% RSLogix 500 project inventoryManagement.RSS, saved by version 8.30.00.16 %
PROJECT "UNTITLED"    % processor: Bul.1763 MicroLogix 1100 Series B %

PROGRAM FILES
  LAD 2   24 rungs

DATA FILES
  O0 OUTPUT  4 elements
  I1 INPUT  6 elements
  S2 STATUS  66 elements
  B3 BINARY  1 elements
  T4 TIMER  1 elements
  C5 COUNTER  1 elements
  R6 CONTROL  1 elements
  N7 INTEGER  9 elements
  F8 FLOAT  1 elements
  ST9 BARCODE  10 elements

LADDER 2
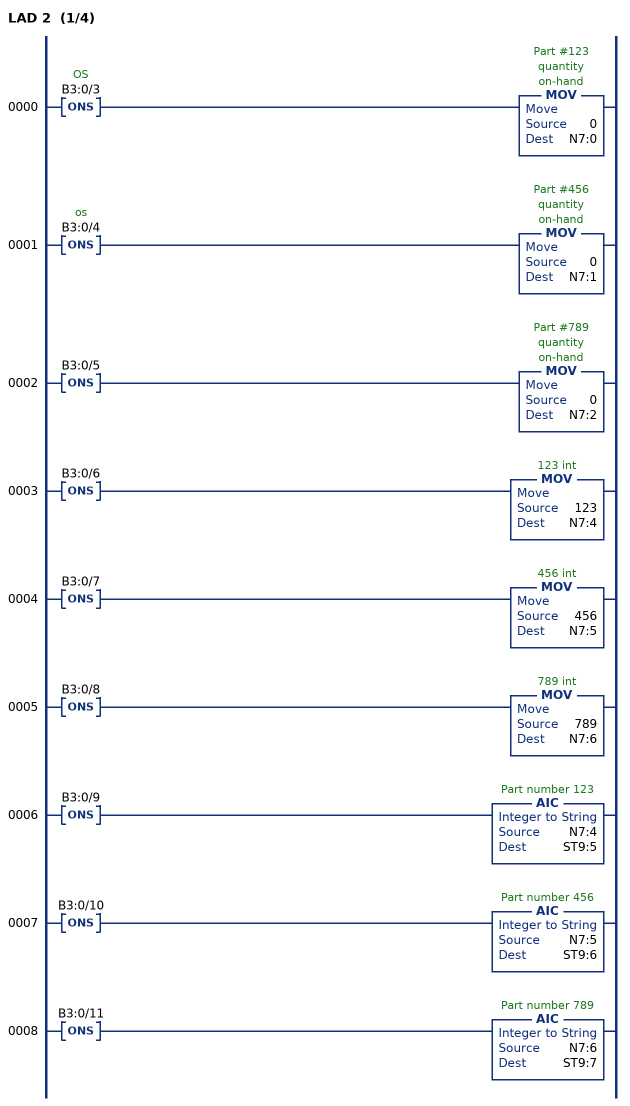
% Rung: 0 %
SOR ONS B3:0/3 MOV 0 N7:0 EOR
%   B3:0/3  "OS" %
%   N7:0  "Part #123 quantity on-hand" %
% Rung: 1 %
SOR ONS B3:0/4 MOV 0 N7:1 EOR
%   B3:0/4  "os" %
%   N7:1  "Part #456 quantity on-hand" %
% Rung: 2 %
SOR ONS B3:0/5 MOV 0 N7:2 EOR
%   N7:2  "Part #789 quantity on-hand" %
% Rung: 3 %
SOR ONS B3:0/6 MOV 123 N7:4 EOR
%   N7:4  "123 int" %
% Rung: 4 %
SOR ONS B3:0/7 MOV 456 N7:5 EOR
%   N7:5  "456 int" %
% Rung: 5 %
SOR ONS B3:0/8 MOV 789 N7:6 EOR
%   N7:6  "789 int" %
% Rung: 6 %
SOR ONS B3:0/9 AIC N7:4 ST9:5 EOR
%   N7:4  "123 int" %
%   ST9:5  "Part number 123" %
% Rung: 7 %
SOR ONS B3:0/10 AIC N7:5 ST9:6 EOR
%   N7:5  "456 int" %
%   ST9:6  "Part number 456" %
% Rung: 8 %
SOR ONS B3:0/11 AIC N7:6 ST9:7 EOR
%   N7:6  "789 int" %
%   ST9:7  "Part number 789" %

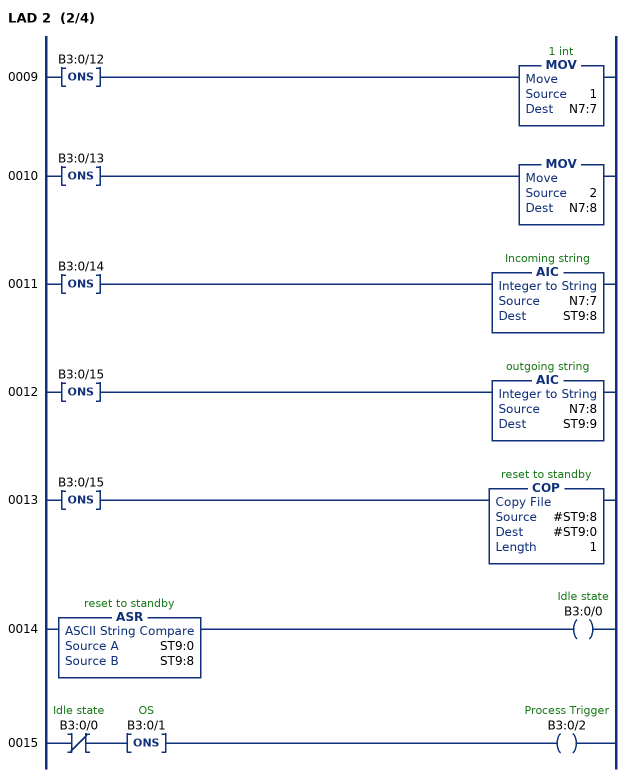
% Rung: 9 %
SOR ONS B3:0/12 MOV 1 N7:7 EOR
%   N7:7  "1 int" %
% Rung: 10 %
SOR ONS B3:0/13 MOV 2 N7:8 EOR
% Rung: 11 %
SOR ONS B3:0/14 AIC N7:7 ST9:8 EOR
%   N7:7  "1 int" %
%   ST9:8  "Incoming string" %
% Rung: 12 %
SOR ONS B3:0/15 AIC N7:8 ST9:9 EOR
%   ST9:9  "outgoing string" %
% Rung: 13 %
SOR ONS B3:0/15 COP #ST9:8 #ST9:0 1 EOR
%   ST9:8  "Incoming string" %
%   ST9:0  "reset to standby" %
% Rung: 14 %
SOR ASR ST9:0 ST9:8 OTE B3:0/0 EOR
%   ST9:0  "reset to standby" %
%   ST9:8  "Incoming string" %
%   B3:0/0  "Idle state" %
% Rung: 15 %
SOR XIO B3:0/0 ONS B3:0/1 OTE B3:0/2 EOR
%   B3:0/0  "Idle state" %
%   B3:0/1  "OS" %
%   B3:0/2  "Process Trigger" %

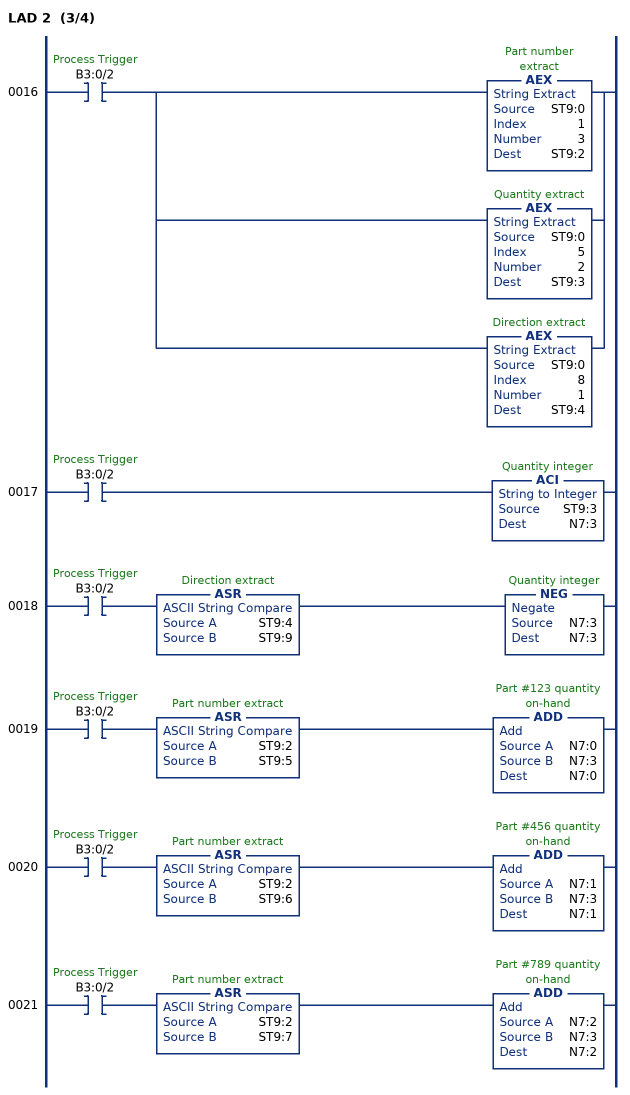
% Rung: 16 %
SOR XIC B3:0/2 BST AEX ST9:0 1 3 ST9:2 NXB BST AEX ST9:0 5 2 ST9:3 NXB AEX ST9:0 8 1 ST9:4 BND BND EOR
%   B3:0/2  "Process Trigger" %
%   ST9:0  "reset to standby" %
%   ST9:2  "Part number extract" %
%   ST9:3  "Quantity extract" %
%   ST9:4  "Direction extract" %
% Rung: 17 %
SOR XIC B3:0/2 ACI ST9:3 N7:3 EOR
%   B3:0/2  "Process Trigger" %
%   ST9:3  "Quantity extract" %
%   N7:3  "Quantity integer" %
% Rung: 18 %
SOR XIC B3:0/2 ASR ST9:4 ST9:9 NEG N7:3 N7:3 EOR
%   B3:0/2  "Process Trigger" %
%   ST9:4  "Direction extract" %
%   ST9:9  "outgoing string" %
%   N7:3  "Quantity integer" %
% Rung: 19 %
SOR XIC B3:0/2 ASR ST9:2 ST9:5 ADD N7:0 N7:3 N7:0 EOR
%   B3:0/2  "Process Trigger" %
%   ST9:2  "Part number extract" %
%   ST9:5  "Part number 123" %
%   N7:0  "Part #123 quantity on-hand" %
%   N7:3  "Quantity integer" %
% Rung: 20 %
SOR XIC B3:0/2 ASR ST9:2 ST9:6 ADD N7:1 N7:3 N7:1 EOR
%   B3:0/2  "Process Trigger" %
%   ST9:2  "Part number extract" %
%   ST9:6  "Part number 456" %
%   N7:1  "Part #456 quantity on-hand" %
%   N7:3  "Quantity integer" %
% Rung: 21 %
SOR XIC B3:0/2 ASR ST9:2 ST9:7 ADD N7:2 N7:3 N7:2 EOR
%   B3:0/2  "Process Trigger" %
%   ST9:2  "Part number extract" %
%   ST9:7  "Part number 789" %
%   N7:2  "Part #789 quantity on-hand" %
%   N7:3  "Quantity integer" %

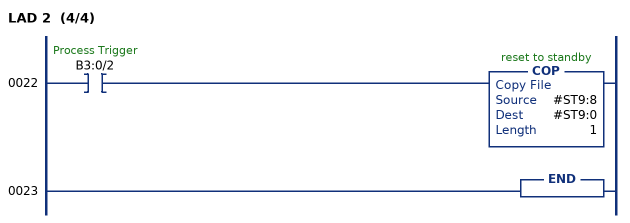
% Rung: 22 %
SOR XIC B3:0/2 COP #ST9:8 #ST9:0 1 EOR
%   B3:0/2  "Process Trigger" %
%   ST9:8  "Incoming string" %
%   ST9:0  "reset to standby" %
% Rung: 23 %
SOR END EOR

OTHER DOCUMENTED ADDRESSES
  ST9:1  STBY
  STANDBY  "Standby hardcode"
